// TIA Portal V16 export
// export: Created 2021-05-26T11:52:20.2864402Z, ExportSetting WithDefaults, DisplayName Totally Integrated Automation Portal, DisplayVersion V16 Update 4, DisplayName TIA Portal Version Control Interface, DisplayVersion V16 Update 2, DisplayName TIA Portal Openness, DisplayVersion V16 Update 4, DisplayName STEP 7 Professional, DisplayVersion V16 Update 4, DisplayName STEP 7 Safety, DisplayVersion V16, DisplayName WinCC Advanced, DisplayVersion V16 Update 4
DATA_BLOCK "COMM_UDP_DB"   // DB3
{ S7_Optimized_Access := 'FALSE'; DB_Accessible_From_OPC_UA := 'FALSE' }
VERSION : 0.1
// stored: AutoNumber false, DBAccessibleFromOPCUA false, IsOnlyStoredInLoadMemory false, IsWriteProtectedInAS false
   VAR
      TSND_BC : Struct
         Start : Bool;
         Busy : Bool;
         Done : Bool;
         Error : Bool;
         Len : UDInt;
         Status : Word;
      END_STRUCT;
      TRCV1_BC : Struct
         Start : Bool;
         Busy : Bool;
         Done : Bool;
         Error : Bool;
         Len : UDInt;
         Status : Word;
      END_STRUCT;
      TRCV2_BC : Struct
         Start : Bool;
         Busy : Bool;
         Done : Bool;
         Error : Bool;
         Len : UDInt;
         Status : Word;
      END_STRUCT;
      TSND_MC1 : Struct
         Start : Bool;
         Busy : Bool;
         Done : Bool;
         Error : Bool;
         Len : UDInt;
         Status : Word;
      END_STRUCT;
      TRCV_MC1 : Struct
         Start : Bool;
         Busy : Bool;
         Done : Bool;
         Error : Bool;
         Len : UDInt;
         Status : Word;
      END_STRUCT;
      TSND_MC2 : Struct
         Start : Bool;
         Busy : Bool;
         Done : Bool;
         Error : Bool;
         Len : UDInt;
         Status : Word;
      END_STRUCT;
      TRCV_MC2 : Struct
         Start : Bool;
         Busy : Bool;
         Done : Bool;
         Error : Bool;
         Len : UDInt;
         Status : Word;
      END_STRUCT;
      TSND_MC3 : Struct
         Start : Bool;
         Busy : Bool;
         Done : Bool;
         Error : Bool;
         Len : UDInt;
         Status : Word;
      END_STRUCT;
      TRCV_MC3 : Struct
         Start : Bool;
         Busy : Bool;
         Done : Bool;
         Error : Bool;
         Len : UDInt;
         Status : Word;
      END_STRUCT;
      TSND_MC4 : Struct
         Start : Bool;
         Busy : Bool;
         Done : Bool;
         Error : Bool;
         Len : UDInt;
         Status : Word;
      END_STRUCT;
      TRCV_MC4 : Struct
         Start : Bool;
         Busy : Bool;
         Done : Bool;
         Error : Bool;
         Len : UDInt;
         Status : Word;
      END_STRUCT;
      TSND_MC5 : Struct
         Start : Bool;
         Busy : Bool;
         Done : Bool;
         Error : Bool;
         Len : UDInt;
         Status : Word;
      END_STRUCT;
      TRCV_MC5 : Struct
         Start : Bool;
         Busy : Bool;
         Done : Bool;
         Error : Bool;
         Len : UDInt;
         Status : Word;
      END_STRUCT;
      TSND_MC6 : Struct
         Start : Bool;
         Busy : Bool;
         Done : Bool;
         Error : Bool;
         Len : UDInt;
         Status : Word;
      END_STRUCT;
      TRCV_MC6 : Struct
         Start : Bool;
         Busy : Bool;
         Done : Bool;
         Error : Bool;
         Len : UDInt;
         Status : Word;
      END_STRUCT;
      TSND_MC7 : Struct
         Start : Bool;
         Busy : Bool;
         Done : Bool;
         Error : Bool;
         Len : UDInt;
         Status : Word;
      END_STRUCT;
      TRCV_MC7 : Struct
         Start : Bool;
         Busy : Bool;
         Done : Bool;
         Error : Bool;
         Len : UDInt;
         Status : Word;
      END_STRUCT;
      TSND_MC8 : Struct
         Start : Bool;
         Busy : Bool;
         Done : Bool;
         Error : Bool;
         Len : UDInt;
         Status : Word;
      END_STRUCT;
      TRCV_MC8 : Struct
         Start : Bool;
         Busy : Bool;
         Done : Bool;
         Error : Bool;
         Len : UDInt;
         Status : Word;
      END_STRUCT;
      TSND_MC9 : Struct
         Start : Bool;
         Busy : Bool;
         Done : Bool;
         Error : Bool;
         Len : UDInt;
         Status : Word;
      END_STRUCT;
      TRCV_MC9 : Struct
         Start : Bool;
         Busy : Bool;
         Done : Bool;
         Error : Bool;
         Len : UDInt;
         Status : Word;
      END_STRUCT;
      TSND_MC10 : Struct
         Start : Bool;
         Busy : Bool;
         Done : Bool;
         Error : Bool;
         Len : UDInt;
         Status : Word;
      END_STRUCT;
      TRCV_MC10 : Struct
         Start : Bool;
         Busy : Bool;
         Done : Bool;
         Error : Bool;
         Len : UDInt;
         Status : Word;
      END_STRUCT;
      TSND_DrvCon : Struct
         Start : Bool;
         Busy : Bool;
         Done : Bool;
         Error : Bool;
         Len : UDInt;
         Status : Word;
      END_STRUCT;
      TRCV_DrvCon : Struct
         Start : Bool;
         Busy : Bool;
         Done : Bool;
         Error : Bool;
         Len : UDInt;
         Status : Word;
      END_STRUCT;
      TSND_FC1 : Struct
         Busy : Bool;
         Done : Bool;
         Error : Bool;
         Len : UDInt;
         Status : Word;
      END_STRUCT;
      TSND_FC2 : Struct
         Busy : Bool;
         Done : Bool;
         Error : Bool;
         Len : UDInt;
         Status : Word;
      END_STRUCT;
      TSND_FC3 : Struct
         Busy : Bool;
         Done : Bool;
         Error : Bool;
         Len : UDInt;
         Status : Word;
      END_STRUCT;
      TSND_FC4 : Struct
         Busy : Bool;
         Done : Bool;
         Error : Bool;
         Len : UDInt;
         Status : Word;
      END_STRUCT;
      TRCV_FC1 : Struct
         Enable : Bool;
         Busy : Bool;
         Done : Bool;
         Error : Bool;
         Len : UDInt;
         Status : Word;
      END_STRUCT;
      TRCV_FC2 : Struct
         Enable : Bool;
         Busy : Bool;
         Done : Bool;
         Error : Bool;
         Len : UDInt;
         Status : Word;
      END_STRUCT;
      TRCV_FC3 : Struct
         Enable : Bool;
         Busy : Bool;
         Done : Bool;
         Error : Bool;
         Len : UDInt;
         Status : Word;
      END_STRUCT;
      TRCV_FC4 : Struct
         Enable : Bool;
         Busy : Bool;
         Done : Bool;
         Error : Bool;
         Len : UDInt;
         Status : Word;
      END_STRUCT;
   END_VAR
BEGIN
END_DATA_BLOCK
